# EPICS IOC start-up script: iocs/vmcIOC/iocBoot/iocvmc/settings.iocsh
# prefix used for all PVs in this IOC
epicsEnvSet("PREFIX", "vmc:")
